         //If Connect requested, start connection establishment
         //---------CONNECT HANDLING-------------
         //--------------------------------------
         IF #tempConnectTrigger OR #tempReconnectTrigger THEN
           IF #statConnectionHdl = 16#0 THEN
             // no connectionHdl is used -> ready to connect
             #statOpcUaRequests.Connect := TRUE;
             // set FB outputs
             #statBusy := TRUE;
             #statStatus := #STATUS_BUSY;
           ELSE
             //connectionHdl might be defect, first delete connectionHdl
             //-> not ready to connect
             #statOpcUaRequests.Disconnect := TRUE;
             //set FB Outputs
             #statBusy := TRUE;
             #statStatus := #STATUS_BUSY;
           END_IF;
         ELSE
           IF #instOpcUaDisconnect.Error OR #instOpcUaDisconnect.Done THEN
             //possibly open connection handle is not available or is disconnected
             //-> ready to connect
             #statOpcUaRequests.Disconnect := FALSE;
             #statOpcUaRequests.Connect := TRUE;
             #statConnectionHdl := 0;
           ELSE
             //nothing done by OPC UA Disconnect block -> Not ready to connect
             #statOpcUaRequests.Connect := FALSE;
           END_IF;
         END_IF;

         //Error at connection establishment
         IF #instOpcUaConnect.Error THEN
           #statError := TRUE;
           #statDone := FALSE;
           #statConnected := FALSE;
           #statErrorId := #ERR_ID_CON;
           #statStatus := #instOpcUaConnect.Status;
         END_IF;

         //Connection establishment was successful
         IF #instOpcUaConnect.Done THEN
           #statConnected := TRUE;
           #statError := FALSE;
           #statErrorId := #ERR_ID_GOOD;
           #statConnectCount += 1;
           #statCase := #CASE_NAMESPACE_GET_INDEX_LIST;
         END_IF;

       END_REGION

     #CASE_NAMESPACE_GET_INDEX_LIST:
       REGION Handle Namespaces
         //Request Namespace get Indexlist
         #statOpcUaRequests.NGIL := TRUE;
         #statStatus := #STATUS_BUSY;

         // Get Index List was not successful
         IF #instOpcUaNamespaceGIL.Error THEN
           //--> Call ConnectionGetStatus if Status = "16#800D0000"
           IF #instOpcUaNamespaceGIL.Status = #STATUS_SERVER_NOT_CONNECTED THEN
             #statCase := #CASE_CONNECTION_GET_STATUS;
           ELSE
             #statCase := #CASE_CONNECT;
           END_IF;
           #statOpcUaRequests.NGIL := FALSE;
           // => OUT
           #statError := TRUE;
           #statBusy := FALSE;
           #statStatus := #instOpcUaNamespaceGIL.Status;
           #statErrorId := #ERR_ID_NGIL;
         END_IF;

         //Get Index List was successful
         IF #instOpcUaNamespaceGIL.Done THEN
           //Check StatusList
           FOR #tempIndex := 0 TO UDINT_TO_INT(CountOfElements(#namespaceUris) - 1) DO
             IF #statOpcUaStatusLists.#NamespaceGIL[#tempIndex] <> 16#0 THEN
               #statOpcUaRequests.NGIL := FALSE;
               // => OUT
               #statError := TRUE;
               #statStatus := #statOpcUaStatusLists.NamespaceGIL[#tempIndex];
               #statErrorId := #ERR_ID_NGIL;
               #statCase := #CASE_CONNECT;
               EXIT;
             END_IF;
           END_FOR;
           #statOpcUaRequests.NGIL := FALSE;
           IF NOT #statError THEN
             //Count up statNamespaceGetIndexCount
             #statNamespaceRegCount += 1;
             //statNamespaceIndexesSet
             #statNamespaceIndexesSet := TRUE;
             // => OUT
             #statError := FALSE;
             #statErrorId := #ERR_ID_GOOD;
             //Next Step
             #statCase := #CASE_NODE_GET_HANDLE_LIST;
           ELSE
             #statCase := #CASE_CONNECTION_GET_STATUS;
           END_IF;
         END_IF;
       END_REGION

     #CASE_NODE_GET_HANDLE_LIST:
       REGION Handle NodeId lists
         //Trigger NodeHandleList SFBs
         IF NOT #statRegisteredWrite AND #writeNodeIds <> NULL AND #writeNodeHdls <> NULL THEN
           #statOpcUaRequests.GHLWrite := TRUE;
           #statStatus := #STATUS_BUSY;
         ELSE
           IF NOT #statRegisteredRead AND #readNodeIds <> NULL AND #readNodeHdls <> NULL THEN
             #statOpcUaRequests.GHLRead := TRUE;
             #statStatus := #STATUS_BUSY;
           ELSE
             IF NOT #statRegisteredMethods AND #methodNodeIds <> NULL AND #methodHdls <> NULL AND #objNodeIds <> NULL THEN
               #statOpcUaRequests.GHLMethods := TRUE;
               #statStatus := #STATUS_BUSY;
             ELSE
               #statCase := #CASE_CONNECTED;
               #statBusy := FALSE;
               #statStatus := #STATUS_IDLE;
             END_IF;
           END_IF;
         END_IF;

         REGION Handle ReadList
           //Read Node Get Handle List was not successful
           IF #InstOpcUaGHLRead.Error THEN
             //--> Call ConnectionGetStatus if Status = "16#800D0000"
             IF #InstOpcUaGHLRead.Status = #STATUS_SERVER_NOT_CONNECTED THEN
               #statCase := #CASE_CONNECTION_GET_STATUS;
             ELSE
               //#statCase := #CASE_CONNECT;
               #statCase := #CASE_CONNECTED;
             END_IF;
             #statOpcUaRequests.GHLRead := FALSE;
             // => OUT
             #statError := TRUE;
             #statStatus := #InstOpcUaGHLRead.Status;
             #statErrorId := #ERR_ID_R_GHL;
           END_IF;

           //Read Node Get Handle List was successful
           IF #InstOpcUaGHLRead.Done THEN
             //Check StatusList
             FOR #tempIndex := 0 TO UDINT_TO_INT(CountOfElements(#readNodeIds) - 1) DO
               IF #statOpcUaStatusLists.#ReadGHL[#tempIndex] <> 16#0 THEN
                 // => OUT
                 #statBusy := FALSE;
                 #statError := TRUE;
                 #statStatus := #statOpcUaStatusLists.#ReadGHL[#tempIndex];
                 #statErrorId := #ERR_ID_R_GHL;
                 //#statCase := #CASE_CONNECT;
                 EXIT;
               END_IF;
             END_FOR;
             #statOpcUaRequests.GHLRead := FALSE;
             // Count up statRegisterCount
             #statRegisterCountRead += 1;
             // Nodes are registered
             #statRegisteredRead := TRUE;
             IF NOT #statError THEN
               // => OUT
               #statError := FALSE;
               #statErrorId := #ERR_ID_GOOD;
             END_IF;
           END_IF;
         END_REGION
         REGION Handle Write List
           //Write Node Get Handle List was not successful
           IF #instOpcUaGHLWrite.Error THEN
             //--> Call ConnectionGetStatus if Status = "16#800D0000"
             IF #instOpcUaGHLWrite.Status = #STATUS_SERVER_NOT_CONNECTED THEN
               #statCase := #CASE_CONNECTION_GET_STATUS;
             ELSE
               //#statCase := #CASE_CONNECT;
               #statCase := #CASE_CONNECTED;
             END_IF;
             #statOpcUaRequests.GHLWrite := FALSE;
             // => OUT
             #statError := TRUE;
             #statStatus := #instOpcUaGHLWrite.Status;
             #statErrorId := #ERR_ID_W_GHL;
           END_IF;

           //Write Node Get Handle List was successful
           IF #instOpcUaGHLWrite.Done THEN
             //Check StatusList
             FOR #tempIndex := 0 TO UDINT_TO_INT(CountOfElements(#writeNodeIds) - 1) DO
               IF #statOpcUaStatusLists.#WriteGHL[#tempIndex] <> 16#0 THEN
                 // => OUT
                 #statBusy := FALSE;
                 #statError := TRUE;
                 #statStatus := #statOpcUaStatusLists.#WriteGHL[#tempIndex];
                 #statErrorId := #ERR_ID_W_GHL;
                 //#statCase := #CASE_CONNECT;
                 EXIT;
               END_IF;
             END_FOR;
             #statOpcUaRequests.GHLWrite := FALSE;
             // Count up statRegisterCount
             #statRegisterCountWrite += 1;
             // Nodes are registered
             #statRegisteredWrite := TRUE;
             IF NOT #statError THEN
               // => OUT
               #statError := FALSE;
               #statErrorId := #ERR_ID_GOOD;
             END_IF;
           END_IF;
         END_REGION

         REGION Handle MethodList
           //Method Get HandleList was not successful
           IF #instOpcUaGHLMethods.Error THEN
             //--> Call ConnectionGetStatus if Status = "16#800D0000"
             IF #instOpcUaGHLMethods.Status = #STATUS_SERVER_NOT_CONNECTED THEN
               #statCase := #CASE_CONNECTION_GET_STATUS;
             ELSE
               //#statCase := #CASE_CONNECT;
               #statCase := #CASE_CONNECTED;
             END_IF;
             #statOpcUaRequests.GHLMethods := FALSE;
             // => OUT
             #statError := TRUE;
             #statStatus := #instOpcUaGHLMethods.Status;
             #statErrorId := #ERR_ID_M_GHL;
           END_IF;

           //Method Get Handle List was successful
           IF #instOpcUaGHLMethods.Done THEN
             //Check StatusList
             FOR #tempIndex := 0 TO UDINT_TO_INT(CountOfElements(#methodNodeIds) - 1) DO
               IF #statOpcUaStatusLists.#MethodGHL[#tempIndex] <> 16#0 THEN
                 // => OUT
                 #statBusy := FALSE;
                 #statError := TRUE;
                 #statStatus := #statOpcUaStatusLists.#MethodGHL[#tempIndex];
                 #statErrorId := #ERR_ID_M_GHL;
                 //#statCase := #CASE_CONNECT;
                 EXIT;
               END_IF;
             END_FOR;
             #statOpcUaRequests.GHLMethods := FALSE;
             // Count up statRegisterCount
             #statRegisterCountMethod += 1;
             // Nodes are registered
             #statRegisteredMethods := TRUE;
             IF NOT #statError THEN
               // => OUT
               #statError := FALSE;
               #statErrorId := #ERR_ID_GOOD;
             END_IF;
           END_IF;
         END_REGION

       END_REGION

     #CASE_CONNECTED:

       REGION Command and Idle
         //Idle as long as no Command was triggered
         IF NOT #statBusy AND NOT #read AND NOT #write AND NOT #callMethod THEN
           #statDone := FALSE;
           #statError := FALSE;
           #statErrorId := #ERR_ID_GOOD;
           #statStatus := #STATUS_IDLE;
         END_IF;
         //OPC_UA_GetStatus function is called cyclically, so the connection is monitored
         #instCycDiag(IN := NOT #statCycDiagTrigger,
                      PT := #CYC_TIME_GCS,
                      Q => #tempCycDiag);
         #statCycDiagTrigger := FALSE;
         IF #tempCycDiag AND NOT #statRHLTrigger THEN
           #statCase := #CASE_CONNECTION_GET_STATUS;
           #statCycDiagTrigger := TRUE;
         END_IF;

         REGION Read
           //Trigger
           IF #statRegisteredRead THEN
             #instReadTrigger(CLK := #read,
                              Q => #tempReadTrigger);
           ELSE
             IF #read THEN
               #statError := TRUE;
               #statErrorId := #ERR_ID_RL;
               #statStatus := #STATUS_NOT_REGISTERED; //Error no ReadList is registerd Request denied
             ELSE
               #statError := FALSE;
               #statErrorId := #ERR_ID_GOOD;
               #statStatus := #STATUS_IDLE; //Error no ReadList is registerd Request denied
             END_IF;
           END_IF;

           IF #tempReadTrigger THEN
             #statOpcUaRequests.Read := TRUE;
             #statBusy := TRUE;
             #statStatus := #STATUS_BUSY;
           ELSE
             #statOpcUaRequests.Read := FALSE;
           END_IF;
           //Error
           IF #instOpcUaReadList.Error THEN
             //--> Call ConnectionGetStatus if Status = "16#800D0000"
             IF #instOpcUaReadList.Status = #STATUS_SERVER_NOT_CONNECTED THEN
               #statCase := #CASE_CONNECTION_GET_STATUS;
             END_IF;
             #statOpcUaRequests.Read := FALSE;
             // => OUT
             #statError := TRUE;
             #statBusy := FALSE;
             #statStatus := #instOpcUaReadList.Status;
             #statErrorId := #ERR_ID_RL;
           END_IF;

           //Done
           IF #instOpcUaReadList.Done THEN
             //Check StatusList
             FOR #tempIndex := 0 TO UDINT_TO_INT(CountOfElements(#readNodeIds) - 1) DO
               IF #statOpcUaStatusLists.#ReadList[#tempIndex] <> 16#0 THEN
                 // => OUT
                 #statError := TRUE;
                 #statDone := FALSE;
                 #statBusy := FALSE;
                 #statStatus := #statOpcUaStatusLists.#ReadList[#tempIndex];
                 #statErrorId := #ERR_ID_RL;
                 EXIT;
               END_IF;
             END_FOR;
             #statOpcUaRequests.Read := FALSE;
             // => OUT
             IF NOT #statError THEN
               #statDone := TRUE;
               #statBusy := FALSE;
               #statError := FALSE;
               #statStatus := #STATUS_DONE;
               #statErrorId := #ERR_ID_GOOD;
               //Count up statReadCount
               #statReadCount += 1;
               //--> Nodes are read continously ...
             END_IF;
           END_IF;
         END_REGION

         REGION Write
           //Trigger
           IF #statRegisteredWrite THEN
             #instWriteTrigger(CLK := #write,
                               Q => #tempWriteTrigger);
           ELSE
             IF #write THEN
               #statError := TRUE;
               #statErrorId := #ERR_ID_WL;
               #statStatus := #STATUS_NOT_REGISTERED; //Error no WriteList is registerd Request denied
             ELSE
               #statError := FALSE;
               #statErrorId := #ERR_ID_GOOD;
               #statStatus := #STATUS_IDLE; //Error no WriteList is registerd Request denied
             END_IF;
           END_IF;

           IF #tempWriteTrigger THEN
             #statOpcUaRequests.Write := TRUE;
             #statBusy := TRUE;
             #statStatus := #STATUS_BUSY;
           ELSE
             #statOpcUaRequests.Write := FALSE;
           END_IF;
           //Error
           IF #instOpcUaWriteList.Error THEN
             //--> Call ConnectionGetStatus if Status = "16#800D0000"
             IF #instOpcUaWriteList.Status = #STATUS_SERVER_NOT_CONNECTED THEN
               #statCase := #CASE_CONNECTION_GET_STATUS;
             END_IF;
             #statOpcUaRequests.Write := FALSE;
             // => OUT
             #statError := TRUE;
             #statBusy := FALSE;
             #statStatus := #instOpcUaWriteList.Status;
             #statErrorId := #ERR_ID_WL;
           END_IF;

           //Done
           IF #instOpcUaWriteList.Done THEN
             //Check StatusList
             FOR #tempIndex := 0 TO UDINT_TO_INT(CountOfElements(#writeNodeIds) - 1) DO
               IF #statOpcUaStatusLists.#WriteList[#tempIndex] <> 16#0 THEN
                 // => OUT
                 #statError := TRUE;
                 #statDone := FALSE;
                 #statBusy := FALSE;
                 #statStatus := #statOpcUaStatusLists.#WriteList[#tempIndex];
                 #statErrorId := #ERR_ID_WL;
                 EXIT;
               END_IF;
             END_FOR;

             #statOpcUaRequests.Write := FALSE;
             // => OUT
             IF NOT #statError THEN
               #statDone := TRUE;
               #statBusy := FALSE;
               #statError := FALSE;
               #statStatus := #STATUS_DONE;
               #statErrorId := #ERR_ID_GOOD;
               //Count up statwriteCount
               #statWriteCount += 1;
               //--> Nodes are write continously ...
             END_IF;
           END_IF;
         END_REGION

         REGION Method Call
           //Trigger
           IF #statRegisteredMethods THEN
             #instMethodCallTrigger(CLK := #callMethod,
                                    Q => #tempMethodCallTrigger);
           ELSE
             IF #callMethod THEN
               #statError := TRUE;
               #statErrorId := #ERR_ID_MC;
               #statStatus := #STATUS_NOT_REGISTERED; //Error no MethodList is registerd Request denied
             ELSE
               #statError := FALSE;
               #statErrorId := #ERR_ID_GOOD;
               #statStatus := #STATUS_IDLE; //Error no MethodList is registerd Request denied
             END_IF;
           END_IF;

           IF #tempMethodCallTrigger THEN
             #statMethodHdlId := #methodHdlIndex * 0;
             //Define statMethodHdl for the input methodHdlIndex choosen index of MethodList
             #tempRetVal := Serialize(SRC_VARIABLE := #methodHdls,
                                      DEST_ARRAY => #statSerializeMethodHdls,
                                      POS := #statMethodHdlId);
             IF #tempRetVal <> 0 THEN
               #statErrorId := #ERR_ID_MC;
               #statStatus := 16#8000 + INT_TO_DWORD(#tempRetVal);
               #statError := TRUE;
             ELSE
               #statMethodHdlId := #methodHdlIndex * 4;
               #statMethodHdl.%B0 := #statSerializeMethodHdls[#statMethodHdlId + 3];
               #statMethodHdl.%B1 := #statSerializeMethodHdls[#statMethodHdlId + 2];
               #statMethodHdl.%B2 := #statSerializeMethodHdls[#statMethodHdlId + 1];
               #statMethodHdl.%B3 := #statSerializeMethodHdls[#statMethodHdlId];
               //Start Method Call
               #statOpcUaRequests.MethodCall := TRUE;
               #statBusy := TRUE;
               #statStatus := #STATUS_BUSY;
             END_IF;
           ELSE
             #statOpcUaRequests.MethodCall := FALSE;
           END_IF;
           //Error
           IF #instOpcUaMethodCall.Error THEN
             //--> Call ConnectionGetStatus if Status = "16#800D0000"
             IF #instOpcUaMethodCall.Status = #STATUS_SERVER_NOT_CONNECTED THEN
               #statCase := #CASE_CONNECTION_GET_STATUS;
             END_IF;
             #statOpcUaRequests.MethodCall := FALSE;
             // => OUT
             #statError := TRUE;
             #statBusy := FALSE;
             #statStatus := #instOpcUaMethodCall.Status;
             #statErrorId := #ERR_ID_MC;
           END_IF;

           //Done
           IF #instOpcUaMethodCall.Done THEN
             //Check MethodResult
             IF #statMethodResult <> 0 THEN
               #statError := TRUE;
               #statBusy := FALSE;
               #statStatus := #statMethodResult;
               #statErrorId := #ERR_ID_MC;
             END_IF;
             #statOpcUaRequests.MethodCall := FALSE;
             // => OUT
             #statDone := TRUE;
             #statBusy := FALSE;
             #statError := FALSE;
             #statStatus := #STATUS_DONE;
             #statErrorId := #ERR_ID_GOOD;
             //Count up statwriteCount
             #statMethodCallCount += 1;
             //--> Methods can be called continously ...
           END_IF;

         END_REGION

         REGION Clear Session 
           #instClearConnTrig(CLK := NOT #connect,
                              Q => #tempRHLTrigger);

           IF #tempRHLTrigger THEN
             #statRHLTrigger := TRUE;
             #statBusy := TRUE;
           END_IF;
           REGION Release lists
             //If Disconnect requested, release nodes -> disconnect established connection
             //-------DISCONNECT HANDLING------------
             //--------------------------------------
             IF #statRHLTrigger THEN
               IF #statRegisteredWrite AND #writeNodeIds <> NULL AND #writeNodeHdls <> NULL THEN
                 #statOpcUaRequests.RHLWrite := TRUE;
                 #statStatus := #STATUS_BUSY;
               ELSE
                 IF #statRegisteredRead AND #readNodeIds <> NULL AND #readNodeHdls <> NULL THEN
                   #statOpcUaRequests.RHLRead := TRUE;
                   #statStatus := #STATUS_BUSY;
                 ELSE
                   IF #statRegisteredMethods AND #methodNodeIds <> NULL AND #methodHdls <> NULL AND #objNodeIds <> NULL THEN
                     #statOpcUaRequests.RHLMethods := TRUE;
                     #statStatus := #STATUS_BUSY;
                   ELSE
                     #statRHLTrigger := FALSE;
                     #statStatus := #STATUS_IDLE;
                   END_IF;
                 END_IF;
               END_IF;
             END_IF;
             REGION Release ReadList
               //Release Handle List of Read Nodes was not successful
               IF #InstOpcUaRHLRead.Error THEN
                 //--> Call ConnectionGetStatus if Status = "16#800D0000"
                 IF #InstOpcUaRHLRead.Status = #STATUS_SERVER_NOT_CONNECTED THEN
                   #statCase := #CASE_CONNECTION_GET_STATUS;
                 END_IF;
                 #statOpcUaRequests.RHLRead := FALSE;
                 // => OUT
                 #statError := TRUE;
                 #statStatus := #InstOpcUaRHLRead.Status;
                 #statErrorId := #ERR_ID_R_RHL;
               END_IF;

               //Release Handle List of Read Nodes was successful
               IF #InstOpcUaRHLRead.Done THEN
                 //Check StatusList
                 FOR #tempIndex := 0 TO UDINT_TO_INT(CountOfElements(#readNodeIds) - 1) DO
                   IF #statOpcUaStatusLists.#ReadRHL[#tempIndex] <> 16#0 THEN
                     // => OUT
                     #statError := TRUE;
                     #statDone := FALSE;
                     #statBusy := FALSE;
                     #statStatus := #statOpcUaStatusLists.#ReadRHL[#tempIndex];
                     #statErrorId := #ERR_ID_R_RHL;
                     EXIT;
                   END_IF;
                 END_FOR;
                 #statOpcUaRequests.RHLRead := FALSE;
                 #statRegisteredRead := FALSE;
                 IF NOT #statError THEN
                   // => OUT
                   #statBusy := FALSE;
                   #statError := FALSE;
                   #statStatus := #STATUS_DONE;
                   #statErrorId := #ERR_ID_GOOD;
                   //--> Nodes are released
                 END_IF;
               END_IF;
             END_REGION

             REGION Release WriteList
               //Release Handle List of Write Nodes was not successful
               IF #instOpcUaRHLWrite.Error THEN
                 //--> Call ConnectionGetStatus if Status = "16#800D0000"
                 IF #instOpcUaRHLWrite.Status = #STATUS_SERVER_NOT_CONNECTED THEN
                   #statCase := #CASE_CONNECTION_GET_STATUS;
                 END_IF;
                 #statOpcUaRequests.RHLWrite := FALSE;
                 // => OUT
                 #statError := TRUE;
                 #statStatus := #instOpcUaRHLWrite.Status;
                 #statErrorId := #ERR_ID_W_RHL;
               END_IF;

               //Release Handle List of Write Nodes was successful
               IF #instOpcUaRHLWrite.Done THEN
                 //Check StatusList
                 FOR #tempIndex := 0 TO UDINT_TO_INT(CountOfElements(#writeNodeIds) - 1) DO
                   IF #statOpcUaStatusLists.WriteRHL[#tempIndex] <> 16#0 THEN
                     // => OUT
                     #statError := TRUE;
                     #statDone := FALSE;
                     #statBusy := FALSE;
                     #statStatus := #statOpcUaStatusLists.#WriteRHL[#tempIndex];
                     #statErrorId := #ERR_ID_W_RHL;
                     EXIT;
                   END_IF;
                 END_FOR;
                 #statOpcUaRequests.RHLWrite := FALSE;
                 #statRegisteredWrite := FALSE;
                 IF NOT #statError THEN
                   // => OUT
                   #statBusy := FALSE;
                   #statError := FALSE;
                   #statStatus := #STATUS_DONE;
                   #statErrorId := #ERR_ID_GOOD;
                   //--> Nodes are released
                 END_IF;
               END_IF;
             END_REGION

             REGION Release MethodList
               //Release Handle List of Methods was not successful
               IF #instOpcUaRHLMethods.Error THEN
                 //--> Call ConnectionGetStatus if Status = "16#800D0000"
                 IF #instOpcUaRHLMethods.Status = #STATUS_SERVER_NOT_CONNECTED THEN
                   #statCase := #CASE_CONNECTION_GET_STATUS;
                 END_IF;
                 #statOpcUaRequests.RHLMethods := FALSE;
                 // => OUT
                 #statError := TRUE;
                 #statStatus := #instOpcUaRHLMethods.Status;
                 #statErrorId := #ERR_ID_M_RHL;
               END_IF;

               //Release Handle List of Methods was successful
               IF #instOpcUaRHLMethods.Done THEN
                 //Check StatusList
                 FOR #tempIndex := 0 TO UDINT_TO_INT(CountOfElements(#methodNodeIds) - 1) DO
                   IF #statOpcUaStatusLists.#MethodRHL[#tempIndex] <> 16#0 THEN
                     // => OUT
                     #statError := TRUE;
                     #statDone := FALSE;
                     #statBusy := FALSE;
                     #statStatus := #statOpcUaStatusLists.#MethodRHL[#tempIndex];
                     #statErrorId := #ERR_ID_M_RHL;
                     EXIT;
                   END_IF;
                 END_FOR;
                 #statOpcUaRequests.RHLMethods := FALSE;
                 #statRegisteredMethods := FALSE;
                 IF NOT #statError THEN
                   // => OUT
                   #statBusy := FALSE;
                   #statError := FALSE;
                   #statStatus := #STATUS_DONE;
                   #statErrorId := #ERR_ID_GOOD;
                   //--> Nodes are released
                 END_IF;
               END_IF;
             END_REGION
           END_REGION

           REGION Disconnect
             #instDisconRTrig(CLK := NOT #statRegisteredRead
                              AND NOT #statRegisteredWrite
                              AND NOT #statRegisteredMethods,
                              //OR (#statConnected AND #statErrorId > 70),
                              Q => #tempDisconnectTrigger);

             IF #tempDisconnectTrigger THEN
               IF #statConnectionHdl <> 16#0 THEN
                 #statOpcUaRequests.Disconnect := TRUE;
                 //set FB Outputs
                 #statBusy := TRUE;
                 #statStatus := #STATUS_BUSY;
                 #statConnectionHdl := 0;
               ELSE
                 #statCase := #CASE_CONNECT;
                 //Error No connection established
               END_IF;
             ELSE
               #statOpcUaRequests.Disconnect := FALSE;
             END_IF;

             //Error at connection establishment
             IF #instOpcUaDisconnect.Error THEN
               #statError := TRUE;
               #statBusy := FALSE;
               #statErrorId := #ERR_ID_DISCON;
               #statStatus := #instOpcUaDisconnect.Status;
               #statCase := #CASE_CONNECTION_GET_STATUS;
             END_IF;

             //Disconnect was successful
             IF #instOpcUaDisconnect.Done THEN
               #statConnected := FALSE;
               #statDone := FALSE;
               #statNamespaceIndexesSet := FALSE;
               #statBusy := FALSE;
               #statOpcUaRequests.Disconnect := FALSE;
               IF #statErrorId <> 0 THEN
                 #statError := TRUE;
               ELSE
                 #statError := FALSE;
                 #statErrorId := #ERR_ID_GOOD;
                 #statStatus := #STATUS_DONE;
               END_IF;
               #statCase := #CASE_CONNECT;
             END_IF;
           END_REGION
         END_REGION
       END_REGION

     #CASE_CONNECTION_GET_STATUS:
       REGION Connection Diagnostics
         #statOpcUaRequests.ConGS := TRUE;
         IF #instOpcUaConnectionGetStatus.Error THEN
           //--> New connection attempt if Status "16#A0000105" (Session could not be reactivated and all resources are cleaned up)
           //or Status "16#80AE_0000" (The network connectoin hs been closed)
           IF #instOpcUaConnectionGetStatus.Status = #STATUS_SESSION_CLEANEDUP OR
             #instOpcUaConnectionGetStatus.Status = #STATUS_BAD_CONNECTION_CLOSED
           THEN
             //Connection is cleaned up
             #statConnected := FALSE;
             #statNamespaceIndexesSet := FALSE; //Namespace Indexes are set via OPC_UA_NamespaceGetIndexList
             #statRegisteredRead := FALSE; //Nodes are not registerd anymore
             #statRegisteredWrite := FALSE; //Nodes are not registerd anymore 
             #statRegisteredMethods := FALSE; //Nodes are not registerd anymore
             //Next Step --> New connection attempt
             #statCase := #CASE_CONNECT;
           END_IF;
           #statOpcUaRequests.ConGS := FALSE;
           // => OUT
           #statError := TRUE;
           #statBusy := FALSE;
           #statStatus := #instOpcUaConnectionGetStatus.Status;
           #statErrorId := #ERR_ID_CON_GS_STATUS;
         END_IF;
         //Done
         IF #instOpcUaConnectionGetStatus.Done THEN
           //ConnectionStatus+ServerState+ServiceLevel are "Good"
           IF #instOpcUaConnectionGetStatus.ConnectionStatus = #UACS_CONNECTED
             AND #instOpcUaConnectionGetStatus.ServerState = #UASS_RUNNING
             AND #instOpcUaConnectionGetStatus.ServiceLevel = #UASL_GOOD
           THEN
             #statOpcUaRequests.ConGS := FALSE;
             //Session is reactivated and nodes are still registered --> Next Step --> CommandAndIdle
             IF #statConnected AND #statNamespaceIndexesSet
               AND (#statRegisteredRead OR #readNodeIds = NULL)
               AND (#statRegisteredWrite OR #writeNodeIds = NULL)
               AND (#statRegisteredMethods OR #methodNodeIds = NULL)
             THEN
               #statBusy := FALSE;
               #statCase := #CASE_CONNECTED;
               //Session is reactivated and nodes are not registered yet --> Next Step --> NodeGetHandleList
             ELSIF #statConnected AND #statNamespaceIndexesSet
               AND (NOT #statRegisteredRead OR NOT #statRegisteredWrite OR NOT #statRegisteredMethods)
             THEN
               #statCase := #CASE_NODE_GET_HANDLE_LIST;
               //Session is reactivated and namespaceIndexes are not set yet --> Next Step --> NamespaceGetIndexList
             ELSIF #statConnected AND NOT #statNamespaceIndexesSet
               AND (NOT #statRegisteredRead OR NOT #statRegisteredWrite OR NOT #statRegisteredMethods)
             THEN
               #statCase := #CASE_NAMESPACE_GET_INDEX_LIST;
               //Session is reactivated (but connected bit isn't set) and namespaceIndexes are set and nodes are registered
               //--> Next Step --> CommandAndIdle
             ELSIF NOT #statConnected AND #statNamespaceIndexesSet
               AND (#statRegisteredRead OR #readNodeIds = NULL)
               AND (#statRegisteredWrite OR #writeNodeIds = NULL)
               AND (#statRegisteredMethods OR #methodNodeIds = NULL)
             THEN
               //connected has to be set
               #statConnected := TRUE;
               #statBusy := FALSE;
               #statRHLTrigger := FALSE;
               #statOpcUaRequests.RHLWrite := FALSE;
               #statOpcUaRequests.RHLRead := FALSE;
               #statOpcUaRequests.RHLMethods := FALSE;
               #statCase := #CASE_CONNECTED;
             END_IF;
           ELSE
             IF #connect THEN
               //ConnectionStatus is not "Good"
               IF #instOpcUaConnectionGetStatus.ConnectionStatus <> #UACS_CONNECTED THEN
                 #statOpcUaRequests.ConGS := FALSE;
                 // => OUT
                 #statError := TRUE;
                 #statBusy := FALSE;
                 #statConnected := FALSE;
                 #statErrorId := #ERR_ID_CON_GS_CSTATE;
                 #statStatus := #instOpcUaConnectionGetStatus.ConnectionStatus;
                 //ServerState is not "Good"
               ELSIF #instOpcUaConnectionGetStatus.ServerState <> #UASS_RUNNING THEN
                 #statOpcUaRequests.ConGS := FALSE;
                 // => OUT
                 #statError := TRUE;
                 #statBusy := FALSE;
                 #statConnected := FALSE;
                 #statStatus := #instOpcUaConnectionGetStatus.ServerState;
                 #statErrorId := #ERR_ID_CON_GS_SSTATE;
                 //ServiceLevel is not "Good"
               ELSIF #instOpcUaConnectionGetStatus.ServiceLevel <> #UASL_GOOD THEN
                 #statOpcUaRequests.ConGS := FALSE;
                 // => OUT
                 #statError := TRUE;
                 #statBusy := FALSE;
                 #statStatus := #instOpcUaConnectionGetStatus.ServiceLevel;
                 #statErrorId := #ERR_ID_CON_GS_SLVL;
               END_IF;
             ELSE
               //connect is not set -> connection was faulty -> back to case CONNECT
               //new connection can be set up
               #statCase := #CASE_CONNECT;
               #statOpcUaRequests.ConGS := FALSE;
               #statRHLTrigger := FALSE;
               #statNamespaceIndexesSet := FALSE;
               #statRegisteredRead := FALSE;
               #statRegisteredWrite := FALSE;
               #statRegisteredMethods := FALSE;
             END_IF;
           END_IF;
         END_IF;
       END_REGION
     ELSE  // Statement section ELSE
       ; //Not reachable
   END_CASE;

   REGION Call SFBs
     //CALL SFB OPC_UA_Connect
     #instOpcUaConnect(REQ := #statOpcUaRequests.Connect,
                       ServerEndpointUrl := #serverEndpointUrl,
                       SessionConnectInfo := #connectionInfo,
                       Timeout := #OPC_UA_FUNCTIONS_TIMEOUT,
                       ConnectionHdl => #statConnectionHdl);

     //CALL SFB OPC_UA_NamespaceGetIndexList 
     #instOpcUaNamespaceGIL(REQ := #statOpcUaRequests.NGIL,
                            ConnectionHdl := #statConnectionHdl,
                            NamespaceUrisCount := UDINT_TO_UINT(CountOfElements(#namespaceUris)),
                            NamespaceUris := #namespaceUris,
                            Timeout := #OPC_UA_FUNCTIONS_TIMEOUT,
                            StatusList := #statOpcUaStatusLists.#NamespaceGIL,
                            NamespaceIndexes := #namespaceIndexes);

     //CALL SFB OPC_UA_NodeGetHandleList_Read
     #InstOpcUaGHLRead(REQ := #statOpcUaRequests.GHLRead,
                       ConnectionHdl := #statConnectionHdl,
                       NodeIDCount := UDINT_TO_UINT(CountOfElements(#readNodeIds)),
                       NodeIDs := #readNodeIds,
                       Timeout := #OPC_UA_FUNCTIONS_TIMEOUT,
                       NamespaceIndexCount := UDINT_TO_UINT(CountOfElements(#namespaceIndexes)),
                       NamespaceIndexes := #namespaceIndexes,
                       NodeStatusList := #statOpcUaStatusLists.#ReadGHL,
                       NodeHdls := #readNodeHdls);

     //CALL SFB OPC_UA_NodeGetHandleList_Write
     #instOpcUaGHLWrite(REQ := #statOpcUaRequests.GHLWrite,
                        ConnectionHdl := #statConnectionHdl,
                        NodeIDCount := UDINT_TO_UINT(CountOfElements(#writeNodeIds)),
                        NodeIDs := #writeNodeIds,
                        Timeout := #OPC_UA_FUNCTIONS_TIMEOUT,
                        NamespaceIndexCount := UDINT_TO_UINT(CountOfElements(#namespaceIndexes)),
                        NamespaceIndexes := #namespaceIndexes,
                        NodeStatusList := #statOpcUaStatusLists.#WriteGHL,
                        NodeHdls := #writeNodeHdls);

     //CALL SFB OPC_UA_MethodGetHandleList
     #instOpcUaGHLMethods(REQ := #statOpcUaRequests.GHLMethods,
                          ConnectionHdl := #statConnectionHdl,
                          NodeIDCount := UDINT_TO_UINT(CountOfElements(#methodNodeIds)),
                          ObjectNodeIDs := #objNodeIds,
                          MethodNodeIDs := #methodNodeIds,
                          Timeout := #OPC_UA_FUNCTIONS_TIMEOUT,
                          NamespaceIndexCount := UDINT_TO_UINT(CountOfElements(#namespaceIndexes)),
                          NamespaceIndexes := #namespaceIndexes,
                          StatusList := #statOpcUaStatusLists.#MethodGHL,
                          MethodHdls := #methodHdls);

     //CALL SFB OPC_UA_ReadList
     #instOpcUaReadList(REQ := #statOpcUaRequests.Read,
                        ConnectionHdl := #statConnectionHdl,
                        NodeHdlCount := UDINT_TO_UINT(CountOfElements(#readNodeHdls)),
                        NodeHdls := #readNodeHdls,
                        Timeout := #OPC_UA_FUNCTIONS_TIMEOUT,
                        NodeStatusList := #statOpcUaStatusLists.#ReadList,
                        TimeStamps := #statOpcUaReadTimeStamps,
                        Variable := #readData);

     //CALL SFB OPC_UA_WriteList
     #instOpcUaWriteList(REQ := #statOpcUaRequests.Write,
                         ConnectionHdl := #statConnectionHdl,
                         NodeHdlCount := UDINT_TO_UINT(CountOfElements(#writeNodeHdls)),
                         NodeHdls := #writeNodeHdls,
                         Timeout := #OPC_UA_FUNCTIONS_TIMEOUT,
                         NodeStatusList := #statOpcUaStatusLists.#WriteList,
                         Variable := #writeData);

     //CALL SFB OPC_UA_MethodCall
     #instOpcUaMethodCall(REQ := #statOpcUaRequests.MethodCall,
                          ConnectionHdl := #statConnectionHdl,
                          MethodHdl := #statMethodHdl,
                          Timeout := #OPC_UA_FUNCTIONS_TIMEOUT,
                          MethodResult := #statMethodResult,
                          InputArguments := #inputArguments,
                          OutputArguments := #outputArguments);

     //CALL SFB OPC_UA_NodeReleaseHandleList_Read
     #InstOpcUaRHLRead(REQ := #statOpcUaRequests.RHLRead,
                       ConnectionHdl := #statConnectionHdl,
                       NodeHdlCount := UDINT_TO_UINT(CountOfElements(#readNodeHdls)),
                       NodeHdls := #readNodeHdls,
                       Timeout := #OPC_UA_FUNCTIONS_TIMEOUT,
                       NodeStatusList := #statOpcUaStatusLists.#ReadRHL);

     //CALL SFB OPC_UA_NodeReleaseHandleList_Write
     #instOpcUaRHLWrite(REQ := #statOpcUaRequests.RHLWrite,
                        ConnectionHdl := #statConnectionHdl,
                        NodeHdlCount := UDINT_TO_UINT(CountOfElements(#writeNodeHdls)),
                        NodeHdls := #writeNodeHdls,
                        Timeout := #OPC_UA_FUNCTIONS_TIMEOUT,
                        NodeStatusList := #statOpcUaStatusLists.#WriteRHL);

     //CALL SFB OPC_UA_MethodReleaseHandleList
     #instOpcUaRHLMethods(REQ := #statOpcUaRequests.RHLMethods,
                          ConnectionHdl := #statConnectionHdl,
                          MethodHdlCount := UDINT_TO_UINT(CountOfElements(#methodHdls)),
                          MethodHdls := #methodHdls,
                          Timeout := #OPC_UA_FUNCTIONS_TIMEOUT,
                          StatusList := #statOpcUaStatusLists.#MethodRHL);

     //CALL SFB OPC_UA_Disconnect
     #instOpcUaDisconnect(REQ := #statOpcUaRequests.Disconnect,
                          ConnectionHdl := #statConnectionHdl,
                          Timeout := #OPC_UA_FUNCTIONS_TIMEOUT);

     //CALL SFB OPC_UA_ConnectionGetStatus
     #instOpcUaConnectionGetStatus(REQ := #statOpcUaRequests.ConGS,
                                   ConnectionHdl := #statConnectionHdl,
                                   Timeout := #OPC_UA_FUNCTIONS_TIMEOUT);
   END_REGION

   REGION Set FB Outputs
     #connected := #statConnected;
     #done := #statDone;
     #busy := #statBusy;
     #errorId := #statErrorId;
     #error := #statError;
     #status := #statStatus;
     #conectionHdl := #statConnectionHdl;
   END_REGION
END_FUNCTION_BLOCK

// ===== library: MasterCopy "OpcUaClient" =====

// folder: OPC UA Client

FUNCTION_BLOCK "OpcUaClient"   // FB2, SCL
TITLE = OpcUaClient
{ S7_Optimized_Access := 'TRUE' }
AUTHOR : SiemensAG
VERSION : 1.0
// OPC UA-Client-Wrapper
   VAR_INPUT
      connect : Bool;
      read : Bool;
      write : Bool;
      callMethod : Bool;
      methodHdlIndex : DInt;
      connectionInfo : OPC_UA_SessionConnectInfo;
      serverEndpointUrl : String;
   END_VAR
   VAR_OUTPUT
      connected : Bool;
      done : Bool;
      busy : Bool;
      error : Bool;
      errorId : Int;
      status : DWord;
      conectionHdl : DWord;
   END_VAR
   VAR_IN_OUT
      namespaceUris : Variant;
      namespaceIndexes : Variant;
      readNodeIds : Variant;
      readNodeHdls : Variant;
      readData : Variant;
      writeNodeIds : Variant;
      writeNodeHdls : Variant;
      writeData : Variant;
      objNodeIds : Variant;
      methodNodeIds : Variant;
      methodHdls : Variant;
      inputArguments : Variant;
      outputArguments : Variant;
   END_VAR
   VAR
      instOpcUaConnect : OPC_UA_Connect;
      instOpcUaConnectionGetStatus : OPC_UA_ConnectionGetStatus;
      instOpcUaNamespaceGIL : OPC_UA_NamespaceGetIndexList;
      InstOpcUaGHLRead : OPC_UA_NodeGetHandleList;
      instOpcUaGHLWrite : OPC_UA_NodeGetHandleList;
      instOpcUaGHLMethods : OPC_UA_MethodGetHandleList;
      InstOpcUaRHLRead : OPC_UA_NodeReleaseHandleList;
      instOpcUaRHLWrite : OPC_UA_NodeReleaseHandleList;
      instOpcUaRHLMethods : OPC_UA_MethodReleaseHandleList;
      instOpcUaReadList : OPC_UA_ReadList;
      instOpcUaWriteList : OPC_UA_WriteList;
      instOpcUaMethodCall : OPC_UA_MethodCall;
      instOpcUaDisconnect : OPC_UA_Disconnect;
      instConnRTrig : R_TRIG;
      instDisconRTrig : R_TRIG;
      instReconTrigger : R_TRIG;
      instNGILTrigger : R_TRIG;
      instReadTrigger : R_TRIG;
      instWriteTrigger : R_TRIG;
      instMethodCallTrigger : R_TRIG;
      instClearConnTrig : R_TRIG;
      statCase : Int;
      statDone : Bool;
      statConnected : Bool;
      statBusy : Bool;
      statError : Bool;
      statErrorId : Int;
      statStatus : DWord;
      statOpcUaRequests : Struct
         Connect : Bool;
         ConGS : Bool;
         NGIL : Bool;
         GHLRead : Bool;
         GHLMethods : Bool;
         GHLWrite : Bool;
         Read : Bool;
         Write : Bool;
         MethodCall : Bool;
         RHLRead : Bool;
         RHLWrite : Bool;
         RHLMethods : Bool;
         Disconnect : Bool;
      END_STRUCT;
      statRHLTrigger : Bool;
      statConnectCount : Int;
      statNamespaceIndexesSet : Bool;
      statNamespaceRegCount : Int;
      statRegisteredRead : Bool;
      statRegisterCountRead : Int;
      statRegisteredWrite : Bool;
      statRegisterCountWrite : Int;
      statRegisteredMethods : Bool;
      statRegisterCountMethod : Int;
      statReadCount : Int;
      statWriteCount : Int;
      statMethodCallCount : DWord;
      statMethodResult : DWord;
      statMethodHdl : DWord;
      statMethodHdlId : DInt;
      statConnectionHdl : DWord;
      instCycDiag : TON_TIME;
      statCycDiagTrigger : Bool;
      statOpcUaReadTimeStamps : Array[0..299] of LDT;
      statSerializeMethodHdls : Array[0..1199] of Byte;
      statOpcUaStatusLists : Struct
         MethodRHL : Array[0..299] of DWord;
         MethodGHL : Array[0..299] of DWord;
         WriteRHL : Array[0..299] of DWord;
         WriteList : Array[0..299] of DWord;
         WriteGHL : Array[0..299] of DWord;
         ReadRHL : Array[0..299] of DWord;
         ReadList : Array[0..299] of DWord;
         ReadGHL : Array[0..299] of DWord;
         NamespaceGIL : Array[0..299] of DWord;
      END_STRUCT;
   END_VAR
   VAR_TEMP
      tempConnectTrigger : Bool;
      tempDisconnectTrigger : Bool;
      tempIndex : Int;
      tempReadTrigger : Bool;
      tempWriteTrigger : Bool;
      tempMethodCallTrigger : Bool;
      tempRetVal : Int;
      tempCycDiag : Bool;
      tempReconnectTrigger : Bool;
      tempRHLTrigger : Bool;
   END_VAR
   VAR CONSTANT
      CASE_CONNECT : Int := 0;
      CASE_NAMESPACE_GET_INDEX_LIST : Int := 1;
      CASE_CONNECTION_GET_STATUS : Int := 2;
      CASE_NODE_GET_HANDLE_LIST : Int := 3;
      CASE_CONNECTED : Int := 4;
      UACS_CONNECTED : UDInt := 0;
      UASS_RUNNING : UDInt := 0;
      UASL_GOOD : UDInt := 16#0000_00FF;
      STATUS_SESSION_CLEANEDUP : DWord := 16#A000_0105;
      STATUS_BUSY : Word := 16#7001;
      STATUS_SERVER_NOT_CONNECTED : DWord := 16#800D_0000;
      STATUS_BAD_CONNECTION_CLOSED : DWord := 16#80AE_0000;
      STATUS_IDLE : Word := 16#7000;
      STATUS_NOT_REGISTERED : Word := 16#80FF;
      STATUS_DONE : Word := 16#0000;
      CYC_TIME_GCS : Time := T#5S;
      OPC_UA_FUNCTIONS_TIMEOUT : Time := T#10S;
      ERR_ID_GOOD : SInt := 0;
      ERR_ID_CON : SInt := 1;
      ERR_ID_CON_GS_STATUS : SInt := 10;
      ERR_ID_CON_GS_CSTATE : SInt := 11;
      ERR_ID_CON_GS_SSTATE : SInt := 12;
      ERR_ID_CON_GS_SLVL : SInt := 13;
      ERR_ID_NGIL : SInt := 2;
      ERR_ID_R_GHL : SInt := 31;
      ERR_ID_W_GHL : SInt := 32;
      ERR_ID_M_GHL : SInt := 33;
      ERR_ID_RL : SInt := 4;
      ERR_ID_WL : SInt := 5;
      ERR_ID_MC : SInt := 6;
      ERR_ID_R_RHL : SInt := 71;
      ERR_ID_W_RHL : SInt := 72;
      ERR_ID_M_RHL : SInt := 73;
      ERR_ID_DISCON : SInt := 8;
   END_VAR
BEGIN
   //=============================================================================
   // Siemens AG (c)Copyright (2019)
   //-----------------------------------------------------------------------------
   // Library: -
   // Tested with: CPU 1513-1 PN;  FW 2.6
   // Engineering: TIA Portal (V15.1)
   // Restrictions: -
   // Requirements: OPC UA Client activated, Fimware V2.6; Set PLC time
   // Functionality: Encapsulates OPC UA client blocks for read, write and method
   //                call including connection handling and diagnosis
   //-----------------------------------------------------------------------------
   // Change log table:
   // Version    Date         Expert in charge           Changes applied
   // 01.00.00   01.02.2019   Siemens SUP Applications   First released version
   //=============================================================================


   //State machine
   CASE #statCase OF
     #CASE_CONNECT:
       REGION Connection Handling
         //initialize FB
         IF NOT #connect THEN
           #statError := FALSE;
           #statBusy := FALSE;
           #statDone := FALSE;
           #statConnected := FALSE;
           #statErrorId := #ERR_ID_GOOD;
           #statStatus := #STATUS_DONE;
         END_IF;

         //Rising Edge detection of connect
         #instConnRTrig(CLK := #connect,
                        Q => #tempConnectTrigger);

         #instReconTrigger(CLK := #connect
                           AND NOT #statConnected
                           AND (#statStatus = #STATUS_SESSION_CLEANEDUP OR #statStatus = #STATUS_BAD_CONNECTION_CLOSED),
                           Q => #tempReconnectTrigger);

         //If Connect requested, start connection establishment
         //---------CONNECT HANDLING-------------
         //--------------------------------------
         IF #tempConnectTrigger OR #tempReconnectTrigger THEN
           IF #statConnectionHdl = 16#0 THEN
             // no connectionHdl is used -> ready to connect
             #statOpcUaRequests.Connect := TRUE;
             // set FB outputs
             #statBusy := TRUE;
             #statStatus := #STATUS_BUSY;
           ELSE
             //connectionHdl might be defect, first delete connectionHdl
             //-> not ready to connect
             #statOpcUaRequests.Disconnect := TRUE;
             //set FB Outputs
             #statBusy := TRUE;
             #statStatus := #STATUS_BUSY;
           END_IF;
         ELSE
           IF #instOpcUaDisconnect.Error OR #instOpcUaDisconnect.Done THEN
             //possibly open connection handle is not available or is disconnected
             //-> ready to connect
             #statOpcUaRequests.Disconnect := FALSE;
             #statOpcUaRequests.Connect := TRUE;
             #statConnectionHdl := 0;
           ELSE
             //nothing done by OPC UA Disconnect block -> Not ready to connect
             #statOpcUaRequests.Connect := FALSE;
           END_IF;
         END_IF;

         //Error at connection establishment
         IF #instOpcUaConnect.Error THEN
           #statError := TRUE;
           #statDone := FALSE;
           #statConnected := FALSE;
           #statErrorId := #ERR_ID_CON;
           #statStatus := #instOpcUaConnect.Status;
         END_IF;

         //Connection establishment was successful
         IF #instOpcUaConnect.Done THEN
           #statConnected := TRUE;
           #statError := FALSE;
           #statErrorId := #ERR_ID_GOOD;
           #statConnectCount += 1;
           #statCase := #CASE_NAMESPACE_GET_INDEX_LIST;
         END_IF;

       END_REGION

     #CASE_NAMESPACE_GET_INDEX_LIST:
       REGION Handle Namespaces
         //Request Namespace get Indexlist
         #statOpcUaRequests.NGIL := TRUE;
         #statStatus := #STATUS_BUSY;

         // Get Index List was not successful
         IF #instOpcUaNamespaceGIL.Error THEN
           //--> Call ConnectionGetStatus if Status = "16#800D0000"
           IF #instOpcUaNamespaceGIL.Status = #STATUS_SERVER_NOT_CONNECTED THEN
             #statCase := #CASE_CONNECTION_GET_STATUS;
           ELSE
             #statCase := #CASE_CONNECT;
           END_IF;
           #statOpcUaRequests.NGIL := FALSE;
           // => OUT
           #statError := TRUE;
           #statBusy := FALSE;
           #statStatus := #instOpcUaNamespaceGIL.Status;
           #statErrorId := #ERR_ID_NGIL;
         END_IF;

         //Get Index List was successful
         IF #instOpcUaNamespaceGIL.Done THEN
           //Check StatusList
           FOR #tempIndex := 0 TO UDINT_TO_INT(CountOfElements(#namespaceUris) - 1) DO
             IF #statOpcUaStatusLists.#NamespaceGIL[#tempIndex] <> 16#0 THEN
               #statOpcUaRequests.NGIL := FALSE;
               // => OUT
               #statError := TRUE;
               #statStatus := #statOpcUaStatusLists.NamespaceGIL[#tempIndex];
               #statErrorId := #ERR_ID_NGIL;
               #statCase := #CASE_CONNECT;
               EXIT;
             END_IF;
           END_FOR;
           #statOpcUaRequests.NGIL := FALSE;
           IF NOT #statError THEN
             //Count up statNamespaceGetIndexCount
             #statNamespaceRegCount += 1;
             //statNamespaceIndexesSet
             #statNamespaceIndexesSet := TRUE;
             // => OUT
             #statError := FALSE;
             #statErrorId := #ERR_ID_GOOD;
             //Next Step
             #statCase := #CASE_NODE_GET_HANDLE_LIST;
           ELSE
             #statCase := #CASE_CONNECTION_GET_STATUS;
           END_IF;
         END_IF;
       END_REGION

     #CASE_NODE_GET_HANDLE_LIST:
       REGION Handle NodeId lists
         //Trigger NodeHandleList SFBs
         IF NOT #statRegisteredWrite AND #writeNodeIds <> NULL AND #writeNodeHdls <> NULL THEN
           #statOpcUaRequests.GHLWrite := TRUE;
           #statStatus := #STATUS_BUSY;
         ELSE
           IF NOT #statRegisteredRead AND #readNodeIds <> NULL AND #readNodeHdls <> NULL THEN
             #statOpcUaRequests.GHLRead := TRUE;
             #statStatus := #STATUS_BUSY;
           ELSE
             IF NOT #statRegisteredMethods AND #methodNodeIds <> NULL AND #methodHdls <> NULL AND #objNodeIds <> NULL THEN
               #statOpcUaRequests.GHLMethods := TRUE;
               #statStatus := #STATUS_BUSY;
             ELSE
               #statCase := #CASE_CONNECTED;
               #statBusy := FALSE;
               #statStatus := #STATUS_IDLE;
             END_IF;
           END_IF;
         END_IF;

         REGION Handle ReadList
           //Read Node Get Handle List was not successful
           IF #InstOpcUaGHLRead.Error THEN
             //--> Call ConnectionGetStatus if Status = "16#800D0000"
             IF #InstOpcUaGHLRead.Status = #STATUS_SERVER_NOT_CONNECTED THEN
               #statCase := #CASE_CONNECTION_GET_STATUS;
             ELSE
               //#statCase := #CASE_CONNECT;
               #statCase := #CASE_CONNECTED;
             END_IF;
             #statOpcUaRequests.GHLRead := FALSE;
             // => OUT
             #statError := TRUE;
             #statStatus := #InstOpcUaGHLRead.Status;
             #statErrorId := #ERR_ID_R_GHL;
           END_IF;

           //Read Node Get Handle List was successful
           IF #InstOpcUaGHLRead.Done THEN
             //Check StatusList
             FOR #tempIndex := 0 TO UDINT_TO_INT(CountOfElements(#readNodeIds) - 1) DO
               IF #statOpcUaStatusLists.#ReadGHL[#tempIndex] <> 16#0 THEN
                 // => OUT
                 #statBusy := FALSE;
                 #statError := TRUE;
                 #statStatus := #statOpcUaStatusLists.#ReadGHL[#tempIndex];
                 #statErrorId := #ERR_ID_R_GHL;
                 //#statCase := #CASE_CONNECT;
                 EXIT;
               END_IF;
             END_FOR;
             #statOpcUaRequests.GHLRead := FALSE;
             // Count up statRegisterCount
             #statRegisterCountRead += 1;
             // Nodes are registered
             #statRegisteredRead := TRUE;
             IF NOT #statError THEN
               // => OUT
               #statError := FALSE;
               #statErrorId := #ERR_ID_GOOD;
             END_IF;
           END_IF;
         END_REGION
         REGION Handle Write List
           //Write Node Get Handle List was not successful
           IF #instOpcUaGHLWrite.Error THEN
             //--> Call ConnectionGetStatus if Status = "16#800D0000"
             IF #instOpcUaGHLWrite.Status = #STATUS_SERVER_NOT_CONNECTED THEN
               #statCase := #CASE_CONNECTION_GET_STATUS;
             ELSE
               //#statCase := #CASE_CONNECT;
               #statCase := #CASE_CONNECTED;
             END_IF;
             #statOpcUaRequests.GHLWrite := FALSE;
             // => OUT
             #statError := TRUE;
             #statStatus := #instOpcUaGHLWrite.Status;
             #statErrorId := #ERR_ID_W_GHL;
           END_IF;

           //Write Node Get Handle List was successful
           IF #instOpcUaGHLWrite.Done THEN
             //Check StatusList
             FOR #tempIndex := 0 TO UDINT_TO_INT(CountOfElements(#writeNodeIds) - 1) DO
               IF #statOpcUaStatusLists.#WriteGHL[#tempIndex] <> 16#0 THEN
                 // => OUT
                 #statBusy := FALSE;
                 #statError := TRUE;
                 #statStatus := #statOpcUaStatusLists.#WriteGHL[#tempIndex];
                 #statErrorId := #ERR_ID_W_GHL;
                 //#statCase := #CASE_CONNECT;
                 EXIT;
               END_IF;
             END_FOR;
             #statOpcUaRequests.GHLWrite := FALSE;
             // Count up statRegisterCount
             #statRegisterCountWrite += 1;
             // Nodes are registered
             #statRegisteredWrite := TRUE;
             IF NOT #statError THEN
               // => OUT
               #statError := FALSE;
               #statErrorId := #ERR_ID_GOOD;
             END_IF;
           END_IF;
         END_REGION

         REGION Handle MethodList
           //Method Get HandleList was not successful
           IF #instOpcUaGHLMethods.Error THEN
             //--> Call ConnectionGetStatus if Status = "16#800D0000"
             IF #instOpcUaGHLMethods.Status = #STATUS_SERVER_NOT_CONNECTED THEN
               #statCase := #CASE_CONNECTION_GET_STATUS;
             ELSE
               //#statCase := #CASE_CONNECT;
               #statCase := #CASE_CONNECTED;
             END_IF;
             #statOpcUaRequests.GHLMethods := FALSE;
             // => OUT
             #statError := TRUE;
             #statStatus := #instOpcUaGHLMethods.Status;
             #statErrorId := #ERR_ID_M_GHL;
           END_IF;

           //Method Get Handle List was successful
           IF #instOpcUaGHLMethods.Done THEN
             //Check StatusList
             FOR #tempIndex := 0 TO UDINT_TO_INT(CountOfElements(#methodNodeIds) - 1) DO
               IF #statOpcUaStatusLists.#MethodGHL[#tempIndex] <> 16#0 THEN
                 // => OUT
                 #statBusy := FALSE;
                 #statError := TRUE;
                 #statStatus := #statOpcUaStatusLists.#MethodGHL[#tempIndex];
                 #statErrorId := #ERR_ID_M_GHL;
                 //#statCase := #CASE_CONNECT;
                 EXIT;
               END_IF;
             END_FOR;
             #statOpcUaRequests.GHLMethods := FALSE;
             // Count up statRegisterCount
             #statRegisterCountMethod += 1;
             // Nodes are registered
             #statRegisteredMethods := TRUE;
             IF NOT #statError THEN
               // => OUT
               #statError := FALSE;
               #statErrorId := #ERR_ID_GOOD;
             END_IF;
           END_IF;
         END_REGION

       END_REGION

     #CASE_CONNECTED:

       REGION Command and Idle
         //Idle as long as no Command was triggered
         IF NOT #statBusy AND NOT #read AND NOT #write AND NOT #callMethod THEN
           #statDone := FALSE;
           #statError := FALSE;
           #statErrorId := #ERR_ID_GOOD;
           #statStatus := #STATUS_IDLE;
         END_IF;
         //OPC_UA_GetStatus function is called cyclically, so the connection is monitored
         #instCycDiag(IN := NOT #statCycDiagTrigger,
                      PT := #CYC_TIME_GCS,
                      Q => #tempCycDiag);
         #statCycDiagTrigger := FALSE;
         IF #tempCycDiag AND NOT #statRHLTrigger THEN
           #statCase := #CASE_CONNECTION_GET_STATUS;
           #statCycDiagTrigger := TRUE;
         END_IF;

         REGION Read
           //Trigger
           IF #statRegisteredRead THEN
             #instReadTrigger(CLK := #read,
                              Q => #tempReadTrigger);
           ELSE
             IF #read THEN
               #statError := TRUE;
               #statErrorId := #ERR_ID_RL;
               #statStatus := #STATUS_NOT_REGISTERED; //Error no ReadList is registerd Request denied
             ELSE
               #statError := FALSE;
               #statErrorId := #ERR_ID_GOOD;
               #statStatus := #STATUS_IDLE; //Error no ReadList is registerd Request denied
             END_IF;
           END_IF;

           IF #tempReadTrigger THEN
             #statOpcUaRequests.Read := TRUE;
             #statBusy := TRUE;
             #statStatus := #STATUS_BUSY;
           ELSE
             #statOpcUaRequests.Read := FALSE;
           END_IF;
           //Error
           IF #instOpcUaReadList.Error THEN
             //--> Call ConnectionGetStatus if Status = "16#800D0000"
             IF #instOpcUaReadList.Status = #STATUS_SERVER_NOT_CONNECTED THEN
               #statCase := #CASE_CONNECTION_GET_STATUS;
             END_IF;
             #statOpcUaRequests.Read := FALSE;
             // => OUT
             #statError := TRUE;
             #statBusy := FALSE;
             #statStatus := #instOpcUaReadList.Status;
             #statErrorId := #ERR_ID_RL;
           END_IF;

           //Done
           IF #instOpcUaReadList.Done THEN
             //Check StatusList
             FOR #tempIndex := 0 TO UDINT_TO_INT(CountOfElements(#readNodeIds) - 1) DO
               IF #statOpcUaStatusLists.#ReadList[#tempIndex] <> 16#0 THEN
                 // => OUT
                 #statError := TRUE;
                 #statDone := FALSE;
                 #statBusy := FALSE;
                 #statStatus := #statOpcUaStatusLists.#ReadList[#tempIndex];
                 #statErrorId := #ERR_ID_RL;
                 EXIT;
               END_IF;
             END_FOR;
             #statOpcUaRequests.Read := FALSE;
             // => OUT
             IF NOT #statError THEN
               #statDone := TRUE;
               #statBusy := FALSE;
               #statError := FALSE;
               #statStatus := #STATUS_DONE;
               #statErrorId := #ERR_ID_GOOD;
               //Count up statReadCount
               #statReadCount += 1;
               //--> Nodes are read continously ...
             END_IF;
           END_IF;
         END_REGION

         REGION Write
           //Trigger
           IF #statRegisteredWrite THEN
             #instWriteTrigger(CLK := #write,
                               Q => #tempWriteTrigger);
           ELSE
             IF #write THEN
               #statError := TRUE;
               #statErrorId := #ERR_ID_WL;
               #statStatus := #STATUS_NOT_REGISTERED; //Error no WriteList is registerd Request denied
             ELSE
               #statError := FALSE;
               #statErrorId := #ERR_ID_GOOD;
               #statStatus := #STATUS_IDLE; //Error no WriteList is registerd Request denied
             END_IF;
           END_IF;

           IF #tempWriteTrigger THEN
             #statOpcUaRequests.Write := TRUE;
             #statBusy := TRUE;
             #statStatus := #STATUS_BUSY;
           ELSE
             #statOpcUaRequests.Write := FALSE;
           END_IF;
           //Error
           IF #instOpcUaWriteList.Error THEN
             //--> Call ConnectionGetStatus if Status = "16#800D0000"
             IF #instOpcUaWriteList.Status = #STATUS_SERVER_NOT_CONNECTED THEN
               #statCase := #CASE_CONNECTION_GET_STATUS;
             END_IF;
             #statOpcUaRequests.Write := FALSE;
             // => OUT
             #statError := TRUE;
             #statBusy := FALSE;
             #statStatus := #instOpcUaWriteList.Status;
             #statErrorId := #ERR_ID_WL;
           END_IF;

           //Done
           IF #instOpcUaWriteList.Done THEN
             //Check StatusList
             FOR #tempIndex := 0 TO UDINT_TO_INT(CountOfElements(#writeNodeIds) - 1) DO
               IF #statOpcUaStatusLists.#WriteList[#tempIndex] <> 16#0 THEN
                 // => OUT
                 #statError := TRUE;
                 #statDone := FALSE;
                 #statBusy := FALSE;
                 #statStatus := #statOpcUaStatusLists.#WriteList[#tempIndex];
                 #statErrorId := #ERR_ID_WL;
                 EXIT;
               END_IF;
             END_FOR;

             #statOpcUaRequests.Write := FALSE;
             // => OUT
             IF NOT #statError THEN
               #statDone := TRUE;
               #statBusy := FALSE;
               #statError := FALSE;
               #statStatus := #STATUS_DONE;
               #statErrorId := #ERR_ID_GOOD;
               //Count up statwriteCount
               #statWriteCount += 1;
               //--> Nodes are write continously ...
             END_IF;
           END_IF;
         END_REGION

         REGION Method Call
           //Trigger
           IF #statRegisteredMethods THEN
             #instMethodCallTrigger(CLK := #callMethod,
                                    Q => #tempMethodCallTrigger);
           ELSE
             IF #callMethod THEN
               #statError := TRUE;
               #statErrorId := #ERR_ID_MC;
               #statStatus := #STATUS_NOT_REGISTERED; //Error no MethodList is registerd Request denied
             ELSE
               #statError := FALSE;
               #statErrorId := #ERR_ID_GOOD;
               #statStatus := #STATUS_IDLE; //Error no MethodList is registerd Request denied
             END_IF;
           END_IF;

           IF #tempMethodCallTrigger THEN
             #statMethodHdlId := #methodHdlIndex * 0;
             //Define statMethodHdl for the input methodHdlIndex choosen index of MethodList
             #tempRetVal := Serialize(SRC_VARIABLE := #methodHdls,
                                      DEST_ARRAY => #statSerializeMethodHdls,
                                      POS := #statMethodHdlId);
             IF #tempRetVal <> 0 THEN
               #statErrorId := #ERR_ID_MC;
               #statStatus := 16#8000 + INT_TO_DWORD(#tempRetVal);
               #statError := TRUE;
             ELSE
               #statMethodHdlId := #methodHdlIndex * 4;
               #statMethodHdl.%B0 := #statSerializeMethodHdls[#statMethodHdlId + 3];
               #statMethodHdl.%B1 := #statSerializeMethodHdls[#statMethodHdlId + 2];
               #statMethodHdl.%B2 := #statSerializeMethodHdls[#statMethodHdlId + 1];
               #statMethodHdl.%B3 := #statSerializeMethodHdls[#statMethodHdlId];
               //Start Method Call
               #statOpcUaRequests.MethodCall := TRUE;
               #statBusy := TRUE;
               #statStatus := #STATUS_BUSY;
             END_IF;
           ELSE
             #statOpcUaRequests.MethodCall := FALSE;
           END_IF;
           //Error
           IF #instOpcUaMethodCall.Error THEN
             //--> Call ConnectionGetStatus if Status = "16#800D0000"
             IF #instOpcUaMethodCall.Status = #STATUS_SERVER_NOT_CONNECTED THEN
               #statCase := #CASE_CONNECTION_GET_STATUS;
             END_IF;
             #statOpcUaRequests.MethodCall := FALSE;
             // => OUT
             #statError := TRUE;
             #statBusy := FALSE;
             #statStatus := #instOpcUaMethodCall.Status;
             #statErrorId := #ERR_ID_MC;
           END_IF;

           //Done
           IF #instOpcUaMethodCall.Done THEN
             //Check MethodResult
             IF #statMethodResult <> 0 THEN
               #statError := TRUE;
               #statBusy := FALSE;
               #statStatus := #statMethodResult;
               #statErrorId := #ERR_ID_MC;
             END_IF;
             #statOpcUaRequests.MethodCall := FALSE;
             // => OUT
             #statDone := TRUE;
             #statBusy := FALSE;
             #statError := FALSE;
             #statStatus := #STATUS_DONE;
             #statErrorId := #ERR_ID_GOOD;
             //Count up statwriteCount
             #statMethodCallCount += 1;
             //--> Methods can be called continously ...
           END_IF;

         END_REGION

         REGION Clear Session 
           #instClearConnTrig(CLK := NOT #connect,
                              Q => #tempRHLTrigger);

           IF #tempRHLTrigger THEN
             #statRHLTrigger := TRUE;
             #statBusy := TRUE;
           END_IF;
           REGION Release lists
             //If Disconnect requested, release nodes -> disconnect established connection
             //-------DISCONNECT HANDLING------------
             //--------------------------------------
             IF #statRHLTrigger THEN
               IF #statRegisteredWrite AND #writeNodeIds <> NULL AND #writeNodeHdls <> NULL THEN
                 #statOpcUaRequests.RHLWrite := TRUE;
                 #statStatus := #STATUS_BUSY;
               ELSE
                 IF #statRegisteredRead AND #readNodeIds <> NULL AND #readNodeHdls <> NULL THEN
                   #statOpcUaRequests.RHLRead := TRUE;
                   #statStatus := #STATUS_BUSY;
                 ELSE
                   IF #statRegisteredMethods AND #methodNodeIds <> NULL AND #methodHdls <> NULL AND #objNodeIds <> NULL THEN
                     #statOpcUaRequests.RHLMethods := TRUE;
                     #statStatus := #STATUS_BUSY;
                   ELSE
                     #statRHLTrigger := FALSE;
                     #statStatus := #STATUS_IDLE;
                   END_IF;
                 END_IF;
               END_IF;
             END_IF;
             REGION Release ReadList
               //Release Handle List of Read Nodes was not successful
               IF #InstOpcUaRHLRead.Error THEN
                 //--> Call ConnectionGetStatus if Status = "16#800D0000"
                 IF #InstOpcUaRHLRead.Status = #STATUS_SERVER_NOT_CONNECTED THEN
                   #statCase := #CASE_CONNECTION_GET_STATUS;
                 END_IF;
                 #statOpcUaRequests.RHLRead := FALSE;
                 // => OUT
                 #statError := TRUE;
                 #statStatus := #InstOpcUaRHLRead.Status;
                 #statErrorId := #ERR_ID_R_RHL;
               END_IF;

               //Release Handle List of Read Nodes was successful
               IF #InstOpcUaRHLRead.Done THEN
                 //Check StatusList
                 FOR #tempIndex := 0 TO UDINT_TO_INT(CountOfElements(#readNodeIds) - 1) DO
                   IF #statOpcUaStatusLists.#ReadRHL[#tempIndex] <> 16#0 THEN
                     // => OUT
                     #statError := TRUE;
                     #statDone := FALSE;
                     #statBusy := FALSE;
                     #statStatus := #statOpcUaStatusLists.#ReadRHL[#tempIndex];
                     #statErrorId := #ERR_ID_R_RHL;
                     EXIT;
                   END_IF;
                 END_FOR;
                 #statOpcUaRequests.RHLRead := FALSE;
                 #statRegisteredRead := FALSE;
                 IF NOT #statError THEN
                   // => OUT
                   #statBusy := FALSE;
                   #statError := FALSE;
                   #statStatus := #STATUS_DONE;
                   #statErrorId := #ERR_ID_GOOD;
                   //--> Nodes are released
                 END_IF;
               END_IF;
             END_REGION

             REGION Release WriteList
               //Release Handle List of Write Nodes was not successful
               IF #instOpcUaRHLWrite.Error THEN
                 //--> Call ConnectionGetStatus if Status = "16#800D0000"
                 IF #instOpcUaRHLWrite.Status = #STATUS_SERVER_NOT_CONNECTED THEN
                   #statCase := #CASE_CONNECTION_GET_STATUS;
                 END_IF;
                 #statOpcUaRequests.RHLWrite := FALSE;
                 // => OUT
                 #statError := TRUE;
                 #statStatus := #instOpcUaRHLWrite.Status;
                 #statErrorId := #ERR_ID_W_RHL;
               END_IF;

               //Release Handle List of Write Nodes was successful
               IF #instOpcUaRHLWrite.Done THEN
                 //Check StatusList
                 FOR #tempIndex := 0 TO UDINT_TO_INT(CountOfElements(#writeNodeIds) - 1) DO
                   IF #statOpcUaStatusLists.WriteRHL[#tempIndex] <> 16#0 THEN
                     // => OUT
                     #statError := TRUE;
                     #statDone := FALSE;
                     #statBusy := FALSE;
                     #statStatus := #statOpcUaStatusLists.#WriteRHL[#tempIndex];
                     #statErrorId := #ERR_ID_W_RHL;
                     EXIT;
                   END_IF;
                 END_FOR;
                 #statOpcUaRequests.RHLWrite := FALSE;
                 #statRegisteredWrite := FALSE;
                 IF NOT #statError THEN
                   // => OUT
                   #statBusy := FALSE;
                   #statError := FALSE;
                   #statStatus := #STATUS_DONE;
                   #statErrorId := #ERR_ID_GOOD;
                   //--> Nodes are released
                 END_IF;
               END_IF;
             END_REGION

             REGION Release MethodList
               //Release Handle List of Methods was not successful
               IF #instOpcUaRHLMethods.Error THEN
                 //--> Call ConnectionGetStatus if Status = "16#800D0000"
                 IF #instOpcUaRHLMethods.Status = #STATUS_SERVER_NOT_CONNECTED THEN
                   #statCase := #CASE_CONNECTION_GET_STATUS;
                 END_IF;
                 #statOpcUaRequests.RHLMethods := FALSE;
                 // => OUT
                 #statError := TRUE;
                 #statStatus := #instOpcUaRHLMethods.Status;
                 #statErrorId := #ERR_ID_M_RHL;
               END_IF;

               //Release Handle List of Methods was successful
               IF #instOpcUaRHLMethods.Done THEN
                 //Check StatusList
                 FOR #tempIndex := 0 TO UDINT_TO_INT(CountOfElements(#methodNodeIds) - 1) DO
                   IF #statOpcUaStatusLists.#MethodRHL[#tempIndex] <> 16#0 THEN
                     // => OUT
                     #statError := TRUE;
                     #statDone := FALSE;
                     #statBusy := FALSE;
                     #statStatus := #statOpcUaStatusLists.#MethodRHL[#tempIndex];
                     #statErrorId := #ERR_ID_M_RHL;
                     EXIT;
                   END_IF;
                 END_FOR;
                 #statOpcUaRequests.RHLMethods := FALSE;
                 #statRegisteredMethods := FALSE;
                 IF NOT #statError THEN
                   // => OUT
                   #statBusy := FALSE;
                   #statError := FALSE;
                   #statStatus := #STATUS_DONE;
                   #statErrorId := #ERR_ID_GOOD;
                   //--> Nodes are released
                 END_IF;
               END_IF;
             END_REGION
           END_REGION

           REGION Disconnect
             #instDisconRTrig(CLK := NOT #statRegisteredRead
                              AND NOT #statRegisteredWrite
                              AND NOT #statRegisteredMethods,
                              //OR (#statConnected AND #statErrorId > 70),
                              Q => #tempDisconnectTrigger);

             IF #tempDisconnectTrigger THEN
               IF #statConnectionHdl <> 16#0 THEN
                 #statOpcUaRequests.Disconnect := TRUE;
                 //set FB Outputs
                 #statBusy := TRUE;
                 #statStatus := #STATUS_BUSY;
                 #statConnectionHdl := 0;
               ELSE
                 #statCase := #CASE_CONNECT;
                 //Error No connection established
               END_IF;
             ELSE
               #statOpcUaRequests.Disconnect := FALSE;
             END_IF;

             //Error at connection establishment
             IF #instOpcUaDisconnect.Error THEN
               #statError := TRUE;
               #statBusy := FALSE;
               #statErrorId := #ERR_ID_DISCON;
               #statStatus := #instOpcUaDisconnect.Status;
               #statCase := #CASE_CONNECTION_GET_STATUS;
             END_IF;

             //Disconnect was successful
             IF #instOpcUaDisconnect.Done THEN
               #statConnected := FALSE;
               #statDone := FALSE;
               #statNamespaceIndexesSet := FALSE;
               #statBusy := FALSE;
               #statOpcUaRequests.Disconnect := FALSE;
               IF #statErrorId <> 0 THEN
                 #statError := TRUE;
               ELSE
                 #statError := FALSE;
                 #statErrorId := #ERR_ID_GOOD;
                 #statStatus := #STATUS_DONE;
               END_IF;
               #statCase := #CASE_CONNECT;
             END_IF;
           END_REGION
         END_REGION
       END_REGION

     #CASE_CONNECTION_GET_STATUS:
       REGION Connection Diagnostics
         #statOpcUaRequests.ConGS := TRUE;
         IF #instOpcUaConnectionGetStatus.Error THEN
           //--> New connection attempt if Status "16#A0000105" (Session could not be reactivated and all resources are cleaned up)
           //or Status "16#80AE_0000" (The network connectoin hs been closed)
           IF #instOpcUaConnectionGetStatus.Status = #STATUS_SESSION_CLEANEDUP OR
             #instOpcUaConnectionGetStatus.Status = #STATUS_BAD_CONNECTION_CLOSED
           THEN
             //Connection is cleaned up
             #statConnected := FALSE;
             #statNamespaceIndexesSet := FALSE; //Namespace Indexes are set via OPC_UA_NamespaceGetIndexList
             #statRegisteredRead := FALSE; //Nodes are not registerd anymore
             #statRegisteredWrite := FALSE; //Nodes are not registerd anymore 
             #statRegisteredMethods := FALSE; //Nodes are not registerd anymore
             //Next Step --> New connection attempt
             #statCase := #CASE_CONNECT;
           END_IF;
           #statOpcUaRequests.ConGS := FALSE;
           // => OUT
           #statError := TRUE;
           #statBusy := FALSE;
           #statStatus := #instOpcUaConnectionGetStatus.Status;
           #statErrorId := #ERR_ID_CON_GS_STATUS;
         END_IF;
         //Done
         IF #instOpcUaConnectionGetStatus.Done THEN
           //ConnectionStatus+ServerState+ServiceLevel are "Good"
           IF #instOpcUaConnectionGetStatus.ConnectionStatus = #UACS_CONNECTED
             AND #instOpcUaConnectionGetStatus.ServerState = #UASS_RUNNING
             AND #instOpcUaConnectionGetStatus.ServiceLevel = #UASL_GOOD
           THEN
             #statOpcUaRequests.ConGS := FALSE;
             //Session is reactivated and nodes are still registered --> Next Step --> CommandAndIdle
             IF #statConnected AND #statNamespaceIndexesSet
               AND (#statRegisteredRead OR #readNodeIds = NULL)
               AND (#statRegisteredWrite OR #writeNodeIds = NULL)
               AND (#statRegisteredMethods OR #methodNodeIds = NULL)
             THEN
               #statBusy := FALSE;
               #statCase := #CASE_CONNECTED;
               //Session is reactivated and nodes are not registered yet --> Next Step --> NodeGetHandleList
             ELSIF #statConnected AND #statNamespaceIndexesSet
               AND (NOT #statRegisteredRead OR NOT #statRegisteredWrite OR NOT #statRegisteredMethods)
             THEN
               #statCase := #CASE_NODE_GET_HANDLE_LIST;
               //Session is reactivated and namespaceIndexes are not set yet --> Next Step --> NamespaceGetIndexList
             ELSIF #statConnected AND NOT #statNamespaceIndexesSet
               AND (NOT #statRegisteredRead OR NOT #statRegisteredWrite OR NOT #statRegisteredMethods)
             THEN
               #statCase := #CASE_NAMESPACE_GET_INDEX_LIST;
               //Session is reactivated (but connected bit isn't set) and namespaceIndexes are set and nodes are registered
               //--> Next Step --> CommandAndIdle
             ELSIF NOT #statConnected AND #statNamespaceIndexesSet
               AND (#statRegisteredRead OR #readNodeIds = NULL)
               AND (#statRegisteredWrite OR #writeNodeIds = NULL)
               AND (#statRegisteredMethods OR #methodNodeIds = NULL)
             THEN
               //connected has to be set
               #statConnected := TRUE;
               #statBusy := FALSE;
               #statRHLTrigger := FALSE;
               #statOpcUaRequests.RHLWrite := FALSE;
               #statOpcUaRequests.RHLRead := FALSE;
               #statOpcUaRequests.RHLMethods := FALSE;
               #statCase := #CASE_CONNECTED;
             END_IF;
           ELSE
             IF #connect THEN
               //ConnectionStatus is not "Good"
               IF #instOpcUaConnectionGetStatus.ConnectionStatus <> #UACS_CONNECTED THEN
                 #statOpcUaRequests.ConGS := FALSE;
                 // => OUT
                 #statError := TRUE;
                 #statBusy := FALSE;
                 #statConnected := FALSE;
                 #statErrorId := #ERR_ID_CON_GS_CSTATE;
                 #statStatus := #instOpcUaConnectionGetStatus.ConnectionStatus;
                 //ServerState is not "Good"
               ELSIF #instOpcUaConnectionGetStatus.ServerState <> #UASS_RUNNING THEN
                 #statOpcUaRequests.ConGS := FALSE;
                 // => OUT
                 #statError := TRUE;
                 #statBusy := FALSE;
                 #statConnected := FALSE;
                 #statStatus := #instOpcUaConnectionGetStatus.ServerState;
                 #statErrorId := #ERR_ID_CON_GS_SSTATE;
                 //ServiceLevel is not "Good"
               ELSIF #instOpcUaConnectionGetStatus.ServiceLevel <> #UASL_GOOD THEN
                 #statOpcUaRequests.ConGS := FALSE;
                 // => OUT
                 #statError := TRUE;
                 #statBusy := FALSE;
                 #statStatus := #instOpcUaConnectionGetStatus.ServiceLevel;
                 #statErrorId := #ERR_ID_CON_GS_SLVL;
               END_IF;
             ELSE
               //connect is not set -> connection was faulty -> back to case CONNECT
               //new connection can be set up
               #statCase := #CASE_CONNECT;
               #statOpcUaRequests.ConGS := FALSE;
               #statRHLTrigger := FALSE;
               #statNamespaceIndexesSet := FALSE;
               #statRegisteredRead := FALSE;
               #statRegisteredWrite := FALSE;
               #statRegisteredMethods := FALSE;
             END_IF;
           END_IF;
         END_IF;
       END_REGION
     ELSE  // Statement section ELSE
       ; //Not reachable
   END_CASE;

   REGION Call SFBs
     //CALL SFB OPC_UA_Connect
     #instOpcUaConnect(REQ := #statOpcUaRequests.Connect,
                       ServerEndpointUrl := #serverEndpointUrl,
                       SessionConnectInfo := #connectionInfo,
                       Timeout := #OPC_UA_FUNCTIONS_TIMEOUT,
                       ConnectionHdl => #statConnectionHdl);

     //CALL SFB OPC_UA_NamespaceGetIndexList 
     #instOpcUaNamespaceGIL(REQ := #statOpcUaRequests.NGIL,
                            ConnectionHdl := #statConnectionHdl,
                            NamespaceUrisCount := UDINT_TO_UINT(CountOfElements(#namespaceUris)),
                            NamespaceUris := #namespaceUris,
                            Timeout := #OPC_UA_FUNCTIONS_TIMEOUT,
                            StatusList := #statOpcUaStatusLists.#NamespaceGIL,
                            NamespaceIndexes := #namespaceIndexes);

     //CALL SFB OPC_UA_NodeGetHandleList_Read
     #InstOpcUaGHLRead(REQ := #statOpcUaRequests.GHLRead,
                       ConnectionHdl := #statConnectionHdl,
                       NodeIDCount := UDINT_TO_UINT(CountOfElements(#readNodeIds)),
                       NodeIDs := #readNodeIds,
                       Timeout := #OPC_UA_FUNCTIONS_TIMEOUT,
                       NamespaceIndexCount := UDINT_TO_UINT(CountOfElements(#namespaceIndexes)),
                       NamespaceIndexes := #namespaceIndexes,
                       NodeStatusList := #statOpcUaStatusLists.#ReadGHL,
                       NodeHdls := #readNodeHdls);

     //CALL SFB OPC_UA_NodeGetHandleList_Write
     #instOpcUaGHLWrite(REQ := #statOpcUaRequests.GHLWrite,
                        ConnectionHdl := #statConnectionHdl,
                        NodeIDCount := UDINT_TO_UINT(CountOfElements(#writeNodeIds)),
                        NodeIDs := #writeNodeIds,
                        Timeout := #OPC_UA_FUNCTIONS_TIMEOUT,
                        NamespaceIndexCount := UDINT_TO_UINT(CountOfElements(#namespaceIndexes)),
                        NamespaceIndexes := #namespaceIndexes,
                        NodeStatusList := #statOpcUaStatusLists.#WriteGHL,
                        NodeHdls := #writeNodeHdls);

     //CALL SFB OPC_UA_MethodGetHandleList
     #instOpcUaGHLMethods(REQ := #statOpcUaRequests.GHLMethods,
                          ConnectionHdl := #statConnectionHdl,
                          NodeIDCount := UDINT_TO_UINT(CountOfElements(#methodNodeIds)),
                          ObjectNodeIDs := #objNodeIds,
                          MethodNodeIDs := #methodNodeIds,
                          Timeout := #OPC_UA_FUNCTIONS_TIMEOUT,
                          NamespaceIndexCount := UDINT_TO_UINT(CountOfElements(#namespaceIndexes)),
                          NamespaceIndexes := #namespaceIndexes,
                          StatusList := #statOpcUaStatusLists.#MethodGHL,
                          MethodHdls := #methodHdls);

     //CALL SFB OPC_UA_ReadList
     #instOpcUaReadList(REQ := #statOpcUaRequests.Read,
                        ConnectionHdl := #statConnectionHdl,
                        NodeHdlCount := UDINT_TO_UINT(CountOfElements(#readNodeHdls)),
                        NodeHdls := #readNodeHdls,
                        Timeout := #OPC_UA_FUNCTIONS_TIMEOUT,
                        NodeStatusList := #statOpcUaStatusLists.#ReadList,
                        TimeStamps := #statOpcUaReadTimeStamps,
                        Variable := #readData);

     //CALL SFB OPC_UA_WriteList
     #instOpcUaWriteList(REQ := #statOpcUaRequests.Write,
                         ConnectionHdl := #statConnectionHdl,
                         NodeHdlCount := UDINT_TO_UINT(CountOfElements(#writeNodeHdls)),
                         NodeHdls := #writeNodeHdls,
                         Timeout := #OPC_UA_FUNCTIONS_TIMEOUT,
                         NodeStatusList := #statOpcUaStatusLists.#WriteList,
                         Variable := #writeData);

     //CALL SFB OPC_UA_MethodCall
     #instOpcUaMethodCall(REQ := #statOpcUaRequests.MethodCall,
                          ConnectionHdl := #statConnectionHdl,
                          MethodHdl := #statMethodHdl,
                          Timeout := #OPC_UA_FUNCTIONS_TIMEOUT,
                          MethodResult := #statMethodResult,
                          InputArguments := #inputArguments,
                          OutputArguments := #outputArguments);

     //CALL SFB OPC_UA_NodeReleaseHandleList_Read
     #InstOpcUaRHLRead(REQ := #statOpcUaRequests.RHLRead,
                       ConnectionHdl := #statConnectionHdl,
                       NodeHdlCount := UDINT_TO_UINT(CountOfElements(#readNodeHdls)),
                       NodeHdls := #readNodeHdls,
                       Timeout := #OPC_UA_FUNCTIONS_TIMEOUT,
                       NodeStatusList := #statOpcUaStatusLists.#ReadRHL);

     //CALL SFB OPC_UA_NodeReleaseHandleList_Write
     #instOpcUaRHLWrite(REQ := #statOpcUaRequests.RHLWrite,
                        ConnectionHdl := #statConnectionHdl,
                        NodeHdlCount := UDINT_TO_UINT(CountOfElements(#writeNodeHdls)),
                        NodeHdls := #writeNodeHdls,
                        Timeout := #OPC_UA_FUNCTIONS_TIMEOUT,
                        NodeStatusList := #statOpcUaStatusLists.#WriteRHL);

     //CALL SFB OPC_UA_MethodReleaseHandleList
     #instOpcUaRHLMethods(REQ := #statOpcUaRequests.RHLMethods,
                          ConnectionHdl := #statConnectionHdl,
                          MethodHdlCount := UDINT_TO_UINT(CountOfElements(#methodHdls)),
                          MethodHdls := #methodHdls,
                          Timeout := #OPC_UA_FUNCTIONS_TIMEOUT,
                          StatusList := #statOpcUaStatusLists.#MethodRHL);

     //CALL SFB OPC_UA_Disconnect
     #instOpcUaDisconnect(REQ := #statOpcUaRequests.Disconnect,
                          ConnectionHdl := #statConnectionHdl,
                          Timeout := #OPC_UA_FUNCTIONS_TIMEOUT);

     //CALL SFB OPC_UA_ConnectionGetStatus
     #instOpcUaConnectionGetStatus(REQ := #statOpcUaRequests.ConGS,
                                   ConnectionHdl := #statConnectionHdl,
                                   Timeout := #OPC_UA_FUNCTIONS_TIMEOUT);
   END_REGION

   REGION Set FB Outputs
     #connected := #statConnected;
     #done := #statDone;
     #busy := #statBusy;
     #errorId := #statErrorId;
     #error := #statError;
     #status := #statStatus;
     #conectionHdl := #statConnectionHdl;
   END_REGION
END_FUNCTION_BLOCK